// TIA Portal V19 export
FUNCTION "FC_FW_Auftrag_Befehl" : Void   // FC187, LAD
{ S7_Optimized_Access := 'TRUE' }
// stored: AutoNumber false, SetENOAutomatically false
   VAR_INPUT
      inQuelle : Int;
      inZiel : Int;
   END_VAR
   VAR_OUTPUT
      Befehl_ok : Bool;
      outQuelle : Int;
      outZiel : Int;
   END_VAR
   VAR_TEMP
      kl_Ziel : Int;
      gr_Ziel : Int;
      Befehl : DWord;
      vor : Bool;
      erlaubt : Bool;
      chk_on : Bool;
      leer : Bool;
   END_VAR
BEGIN

REGION Network 1 (SCL)
   #Befehl_ok := FALSE;
   #outQuelle := 0;
   #outZiel := 0;

   #vor := #inZiel >= #inQuelle;
   #leer := #inZiel = 0;

   IF #leer THEN
       #kl_Ziel := #inZiel;
       #gr_Ziel := #inZiel;
   ELSIF #vor THEN
       #kl_Ziel := #inQuelle;
       #gr_Ziel := #inZiel;
   ELSE
       #kl_Ziel := #inZiel;
       #gr_Ziel := #inQuelle;
   END_IF;

   #chk_on := FALSE;// ("DB_POS".POS[#inQuelle].WT_DB <> 0) AND "DB_POS".POS[#inQuelle].fertig;

   IF NOT #leer THEN
       IF ("DB_POS".POS[#inQuelle].next_WT = 0) OR NOT "DB_POS".POS[#inQuelle].belegt THEN
           RETURN;
       END_IF;

       IF "DB_POS".POS[#inQuelle].Quelle OR "DB_POS".POS[#inQuelle].Sperre_out OR "DB_POS".POS[#inQuelle].notFG_out THEN
           RETURN;
       END_IF;

       IF ("DB_POS".POS[#inZiel].next_WT <> "DB_POS".POS[#inQuelle].next_WT) THEN
           IF ("DB_POS".POS[#inZiel].next_WT <> 0) OR "DB_POS".POS[#inZiel].belegt THEN
               RETURN;
           END_IF;
       END_IF;

       IF "DB_POS".POS[#inZiel].Ziel OR "DB_POS".POS[#inZiel].Sperre_in OR "DB_POS".POS[#inZiel].notFG_in THEN
           RETURN;
       END_IF;

   END_IF;

   "FC_FW_Befehl_ok"(FW_Nr:=1,
                     kl_Z:=#kl_Ziel,
                     Gr_Z:=#gr_Ziel,
                     QT_Check:=TRUE,
                     Ablassen:=FALSE,
                     vor:=#vor,
                     chk_on:=#chk_on,
                     erlaubt=>#erlaubt);

   IF NOT #erlaubt OR NOT "DI_FW_1".ZST.BEREIT THEN
       RETURN;
   END_IF;

   IF #leer THEN
       #Befehl := dw#16#F0010000;
   ELSE
       #Befehl := dw#16#F0030000;
   END_IF;

   #Befehl := #Befehl OR SHL_INT(IN:=#inQuelle,N:=8) OR #inZiel;
   "DI_FW_1".ZST.BEFEHL := #Befehl;

   #Befehl_ok := TRUE;
   #outQuelle := #inQuelle;
   #outZiel := #inZiel;
END_REGION
END_FUNCTION
